// TIA Portal V20 export
TYPE "LKinCtrl_typeApproachPoint"
// stored: Access Published
   STRUCT
      trigger { ExternalAccessible := 'False'; ExternalVisible := 'False'; ExternalWritable := 'False'} : Bool;
      point { ExternalAccessible := 'False'; ExternalVisible := 'False'; ExternalWritable := 'False'} : "LKinCtrl_typePoint";
   END_STRUCT;
END_TYPE
